(* PLC project test_ethercat, Laurent BESSARD test_ethercat 1.0 *)
(* stored: creationDateTime 2011-10-20T19:01:52, modificationDateTime 2012-03-31T16:16:33 *)

PROGRAM Prog
  VAR
    CLOCK AT %QX0.0.2.28672.1 : BOOL;
    LED AT %QX0.0.2.28688.1 : BOOL := TRUE;
    ControlWord AT %QW0.0.3.24640.0 : UINT;
    StatusWord AT %IW0.0.3.24641.0 : UINT;
    ErrorCode AT %IW0.0.3.24639.0 : UINT;
    ModeDisplay AT %IB0.0.3.24673.0 : SINT;
    ActualPosition AT %ID0.0.3.24676.0 : DINT;
    TargetPosition AT %QD0.0.3.24698.0 : DINT;
  END_VAR

CLOCK := NOT CLOCK;
          
END_PROGRAM

PROGRAM test_MCL
  VAR
    CLOCK : UDINT;
  END_VAR
  VAR
    Axis AT %IW0.0.3.0 : AXIS_REF;
  END_VAR
  VAR
    switch : MC_Power;
    move1 : MC_MoveAbsolute;
  END_VAR

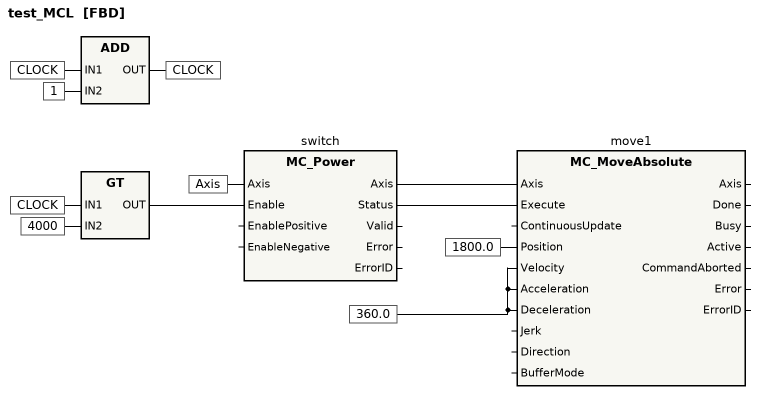
(* FBD diagram, written out as Structured Text *)
CLOCK := CLOCK + 1;
switch(Axis := Axis, Enable := CLOCK > 4000);
move1(Axis := switch.Axis, Execute := switch.Status, Position := 1800.0, Velocity := 360.0, Acceleration := 360.0, Deceleration := 360.0);
END_PROGRAM

CONFIGURATION conf
  RESOURCE res ON PLC
    TASK main_task(INTERVAL := T#0.5ms, PRIORITY := 0);
    PROGRAM main_instance WITH main_task : Prog;
    PROGRAM test_MCL_instance WITH main_task : test_MCL;
  END_RESOURCE
END_CONFIGURATION
